Yaskawa INFORM job: P_XR.JBI

/JOB
//NAME P_XR
///FOLDERNAME INNE
//POS
///NPOS 7,7,7,0,0,0
///TOOL 0
///POSTYPE PULSE
///PULSE
C00000=21,4464,50400,25423,61768,35535
C00001=3981,5204,51584,48389,65423,32215
C00002=12650,-2127,36901,76202,72057,31688
C00003=17586,-13128,12912,74400,71362,36388
C00004=-8487,1038,43440,-9791,61422,40030
C00005=-11449,-2648,35921,-31605,63771,42978
C00006=-14523,-9402,21672,-59597,69425,45285
BC00000=103636,1063121,678632
BC00001=103636,1063121,678632
BC00002=103636,1063121,678632
BC00003=103636,1063121,678632
BC00004=103636,1063121,678632
BC00005=103636,1063121,678632
BC00006=103636,1063121,678632
EC00000=0,0
EC00001=-167491,0
EC00002=-431280,0
EC00003=-525386,0
EC00004=274969,0
EC00005=440232,0
EC00006=678625,0
//INST
///DATE 2023/10/04 15:13
///ATTR SC,RW
///GROUP1 RB1,BS1
///GROUP2 ST1
NOP
MOVJ C00000 BC00000 VJ=0.78  +MOVJ EC00000 VJ=0.78
MOVJ C00001 BC00001 VJ=0.78  +MOVJ EC00001 VJ=0.78
MOVJ C00002 BC00002 VJ=0.78  +MOVJ EC00002 VJ=0.78
MOVJ C00003 BC00003 VJ=0.78  +MOVJ EC00003 VJ=0.78
MOVJ C00004 BC00004 VJ=0.78  +MOVJ EC00004 VJ=0.78
MOVJ C00005 BC00005 VJ=0.78  +MOVJ EC00005 VJ=0.78
MOVJ C00006 BC00006 VJ=0.78  +MOVJ EC00006 VJ=0.78
END
